FUNCTION F_CalcPfeifferCheckSum : BYTE
VAR_INPUT
    sData: STRING;
END_VAR
VAR
    bSum: BYTE;
    i: INT;
END_VAR

bSum := 0;

FOR i := 1 TO LEN(sData) DO
    bSum := bSum + F_ToASC(MID(sData,1,i));
END_FOR

F_CalcPfeifferChecksum := bSum;

END_FUNCTION

(* stored: Version 1.1.0.1
   POU F_CalcPfeifferCheckSum: Id {16130ab7-d093-4369-b333-020b7bba7100}, SpecialFunc None *)
